TEXTLIST nPlcEventTableHeader
  0 = 'Tip' | English: 'Event Type' | Turkish: 'Tip'
  1 = 'Mesaj' | English: 'Event' | Turkish: 'Mesaj'
  2 = 'Zaman' | English: 'Event Time' | Turkish: 'Zaman'
  3 = 'Onay' | English: 'Ack Time' | Turkish: 'Onay'
   = ''
END_TEXTLIST

(* stored: Version 1.1.0.1, ProductVersion 3.1.4024.6
   TextList nPlcEventTableHeader: Id {61529483-731f-437e-8ad6-d12f8e0b5305} *)
